// TwinCAT 3 PLC project PartDispencerPLC
// ProgramVersion: 3.1.4023.0
// libraries:
//   Tc2_MC2, * (Beckhoff Automation GmbH)
//   Tc2_NC, * (Beckhoff Automation GmbH)
//   Tc2_Standard, * (Beckhoff Automation GmbH)
//   Tc2_System, * (Beckhoff Automation GmbH)
//   Tc3_Module, * (Beckhoff Automation GmbH)
// project tree:
//   DUTs/ ST_StationControls.TcDUT
//   GVLs/ Globals.TcGVL, IO.TcGVL
//   / PlcTask.TcTTO
//   POUs/Conveyor/ FB_Conveyor.TcPOU
//   POUs/ MAIN.TcPOU
//   POUs/StationBin/ FB_StationBin.TcPOU
// real-time tasks:
//   TASK PlcTask: cycle T#10ms, priority 20, ADS port 350
// motion (NC):
//   TASK NC-Task 1 SAF: cycle T#2ms, priority 4, ADS port 501
//   TASK NC-Task 1 SVB: cycle T#10ms, priority 8, ADS port 511
//   AXIS Axis Ref (id 1)
//     OtherSettings: AllowMotionCmdToSlave=true
//     encoder EncType=4
//       EncPara: MaxCount=#x0000ffff
//         Inc: RefSoftSyncMask=#x0000ffff
//     drive DrvType=5
//       Analog: TorqueSetpointScale=10, ScaleFactorActTorque=0.1
//       TimeComp: TaskDelayCycles=1
//     controller CtrType=1
//       CtrPara: PriorControlFactor=1
//         Observer: BandWidth=20
// I/O:
//   DEVICE Device 1 (EtherCAT) (disabled), AmsNetId 192.168.0.103.2.1
//     Term 1 (EK1100) [EK1100 EtherCAT Coupler (2A E-Bus)]
//       Term 2 (EL1809) [EL1809 16Ch. Dig. Input 24V, 3ms]
//       Term 3 (EL1809) [EL1809 16Ch. Dig. Input 24V, 3ms]
//       Term 4 (EL2809) [EL2809 16Ch. Dig. Output 24V, 0.5A]
//       Term 5 (EL2809) [EL2809 16Ch. Dig. Output 24V, 0.5A]
//       Term 6 (EL2521) [EL2521 1Ch. Pulse Train Output]
// variable links:
//   NC-Task 1 SAF/Axes/Axis Ref <-> Device 1 (EtherCAT)/Term 1 (EK1100)/Term 6 (EL2521)
//     Drive/Inputs/In/nState1 @bit 6 <-> PTO Status/Status/Error
//     Drive/Inputs/In/nState1 @bit 1 <-> PTO Status/Status/Ramp active
//     Drive/Inputs/In/nState1 <-> PTO Status/Status/Sel. Ack/End counter
//     Drive/Inputs/In/nState1 @bit 4 <-> PTO Status/Status/Status of input target
//     Drive/Inputs/In/nState1 @bit 5 <-> PTO Status/Status/Status of input zero
//     Drive/Inputs/In/nState2 @bit 5 <-> PTO Status/Status/Sync error
//     Drive/Inputs/In/nState2 @bit 7 <-> PTO Status/Status/TxPDO Toggle
//     Drive/Inputs/In/nState4 @bit 1 <-> WcState/InputToggle
//     Drive/Inputs/In/nState4 <-> WcState/WcState
//     Drive/Outputs/Out/nCtrl1 @bit 1 <-> PTO Control/Control/Disable ramp
//     Drive/Outputs/Out/nCtrl1 <-> PTO Control/Control/Frequency select
//     Drive/Outputs/Out/nCtrl1 @bit 2 <-> PTO Control/Control/Go counter
//     Drive/Outputs/Out/nDataOut1[0] <-> PTO Control/Frequency value
//     Drive/Outputs/Out/nDataOut5 <-> PTO Target compact/Target counter value
//     Enc/Inputs/In/nDataIn1[0] <-> ENC Status compact/Counter value
//     Enc/Inputs/In/nState1 @bit 4 <-> ENC Status compact/Status/Counter overflow
//     Enc/Inputs/In/nState1 @bit 3 <-> ENC Status compact/Status/Counter underflow
//     Enc/Inputs/In/nState1 @bit 2 <-> ENC Status compact/Status/Set counter done
//     Enc/Inputs/In/nState2 @bit 5 <-> ENC Status compact/Status/Sync error
//     Enc/Inputs/In/nState2 @bit 7 <-> ENC Status compact/Status/TxPDO Toggle
//     Enc/Inputs/In/nState4 @bit 1 <-> WcState/InputToggle
//     Enc/Inputs/In/nState4 <-> WcState/WcState
//     Enc/Outputs/Out/nCtrl1 @bit 2 <-> ENC Control compact/Control/Set counter
//     Enc/Outputs/Out/nDataOut1[0] <-> ENC Control compact/Set counter value
//   PartDispencerPLC/PartDispencerPLC Instance <-> Device 1 (EtherCAT)/Term 1 (EK1100)/Term 2 (EL1809)
//     PlcTask Inputs/IO.iBowl_present_sensor_on_clamp <-> Channel 16/Input
//     PlcTask Inputs/IO.iStation_1_1_Dispense_Sensor <-> Channel 3/Input
//     PlcTask Inputs/IO.iStation_1_2_Dispense_Sensor <-> Channel 6/Input
//     PlcTask Inputs/IO.iStation_1_3_Dispense_Sensor <-> Channel 9/Input
//     PlcTask Inputs/IO.iStation_2_1_Dispense_Sensor <-> Channel 12/Input
//     PlcTask Inputs/IO.iStation_2_2_Dispense_Sensor <-> Channel 15/Input
//     PlcTask Inputs/IO.iStation_1_1_Home_Sensor <-> Channel 1/Input
//     PlcTask Inputs/IO.iStation_1_2_Home_Sensor <-> Channel 4/Input
//     PlcTask Inputs/IO.iStation_1_3_Home_Sensor <-> Channel 7/Input
//     PlcTask Inputs/IO.iStation_2_1_Home_Sensor <-> Channel 10/Input
//     PlcTask Inputs/IO.iStation_2_2_Home_Sensor <-> Channel 13/Input
//     PlcTask Inputs/IO.iStation_1_1_Safe_Sensor <-> Channel 2/Input
//     PlcTask Inputs/IO.iStation_1_2_Safe_Sensor <-> Channel 5/Input
//     PlcTask Inputs/IO.iStation_1_3_Safe_Sensor <-> Channel 8/Input
//     PlcTask Inputs/IO.iStation_2_1_Safe_Sensor <-> Channel 11/Input
//     PlcTask Inputs/IO.iStation_2_2_Safe_Sensor <-> Channel 14/Input
//   PartDispencerPLC/PartDispencerPLC Instance <-> Device 1 (EtherCAT)/Term 1 (EK1100)/Term 3 (EL1809)
//     PlcTask Inputs/IO.iBowl_10_percent_full <-> Channel 10/Input
//     PlcTask Inputs/IO.iBowl_25_percent_full <-> Channel 9/Input
//     PlcTask Inputs/IO.iBowl_50_percent_full <-> Channel 8/Input
//     PlcTask Inputs/IO.iConveyor_Home_Sensor <-> Channel 4/Input
//     PlcTask Inputs/IO.iConveyor_Position_1_Sensor <-> Channel 5/Input
//     PlcTask Inputs/IO.iConveyor_Position_2_Sensor <-> Channel 6/Input
//     PlcTask Inputs/IO.iConveyor_Position_3_Sensor <-> Channel 7/Input
//     PlcTask Inputs/IO.iStation_1_1_Part_Present_Sensor <-> Channel 11/Input
//     PlcTask Inputs/IO.iStation_1_2_Part_Present_Sensor <-> Channel 12/Input
//     PlcTask Inputs/IO.iStation_1_3_Part_Present_Sensor <-> Channel 13/Input
//     PlcTask Inputs/IO.iStation_2_1_Part_Present_Sensor <-> Channel 14/Input
//     PlcTask Inputs/IO.iStation_2_2_Part_Present_Sensor <-> Channel 15/Input
//     PlcTask Inputs/IO.iStation_2_3_Part_Present_Sensor <-> Channel 16/Input
//     PlcTask Inputs/IO.iStation_2_3_Dispense_Sensor <-> Channel 3/Input
//     PlcTask Inputs/IO.iStation_2_3_Home_Sensor <-> Channel 1/Input
//     PlcTask Inputs/IO.iStation_2_3_Safe_Sensor <-> Channel 2/Input
//   PartDispencerPLC/PartDispencerPLC Instance <-> Device 1 (EtherCAT)/Term 1 (EK1100)/Term 4 (EL2809)
//     PlcTask Outputs/IO.oDirection_OF_Driver_1 <-> Channel 2/Output
//     PlcTask Outputs/IO.oDirection_of_Driver_{2..5} <-> Channel {5..14 step 3}/Output  (4 links)
//     PlcTask Outputs/IO.oEnable_of_Driver_{1..5} <-> Channel {3..15 step 3}/Output  (5 links)
//     PlcTask Outputs/IO.oR{1..5}_NO_Contact <-> Channel {1..13 step 3}/Output  (5 links)
//     PlcTask Outputs/IO.oSPARE_1 <-> Channel 16/Output
//   PartDispencerPLC/PartDispencerPLC Instance <-> Device 1 (EtherCAT)/Term 1 (EK1100)/Term 5 (EL2809)
//     PlcTask Outputs/IO.oDirection_OF_Driver_6 <-> Channel 2/Output
//     PlcTask Outputs/IO.oDirection_of_Driver_7 <-> Channel 5/Output
//     PlcTask Outputs/IO.oDirection_of_Driver_8 <-> Channel 8/Output
//     PlcTask Outputs/IO.oEnable_of_Driver_6 <-> Channel 3/Output
//     PlcTask Outputs/IO.oEnable_of_Driver_7 <-> Channel 6/Output
//     PlcTask Outputs/IO.oEnable_of_Driver_8 <-> Channel 9/Output
//     PlcTask Outputs/IO.oR6_NO_Contact <-> Channel 1/Output
//     PlcTask Outputs/IO.oR7_NO_Contact <-> Channel 4/Output
//     PlcTask Outputs/IO.oR8_NO_Contact <-> Channel 7/Output
//     PlcTask Outputs/IO.oSPARE_{5..11} <-> Channel {10..16}/Output  (7 links)

CONFIGURATION PartDispencerPLC
    RESOURCE PLC ON TwinCAT3
        TASK PlcTask(INTERVAL := T#10ms, PRIORITY := 20);
        PROGRAM MAIN WITH PlcTask : MAIN;
    END_RESOURCE
END_CONFIGURATION

// ---- DUTs/ST_StationControls.TcDUT
TYPE ST_StationControls :
STRUCT
	bEnable			: BOOL;
	bReset			: BOOL;
	bError			: BOOL;
	sStatus			: STRING(255);
END_STRUCT
END_TYPE

// ---- GVLs/Globals.TcGVL
{attribute 'qualified_only'}
VAR_GLOBAL
	ConveyorControl			:ST_StationControls;
	
	Bin1Control				:ST_StationControls;
	Bin2Control				:ST_StationControls;
	Bin3Control				:ST_StationControls;
	Bin4Control				:ST_StationControls;
	Bin5Control				:ST_StationControls;
	Bin6Control				:ST_StationControls;
	
	bResetPartCount_Station1	: BOOL := FALSE;
	bResetPartCount_Station2	: BOOL := FALSE;
	
	axisRef						: AXIS_REF;
END_VAR

// ---- GVLs/IO.TcGVL
{attribute 'qualified_only'}
VAR_GLOBAL
// ======================== Inputs ==================================
	// SLOT 1 - EL1809
	iStation_1_1_Home_Sensor				AT %I* :BOOL;
	iStation_1_1_Safe_Sensor             	AT %I* :BOOL;
	iStation_1_1_Dispense_Sensor         	AT %I* :BOOL;
	iStation_1_2_Home_Sensor             	AT %I* :BOOL;
	iStation_1_2_Safe_Sensor             	AT %I* :BOOL;
	iStation_1_2_Dispense_Sensor         	AT %I* :BOOL;
	iStation_1_3_Home_Sensor             	AT %I* :BOOL;
	iStation_1_3_Safe_Sensor             	AT %I* :BOOL;
	iStation_1_3_Dispense_Sensor         	AT %I* :BOOL;
	iStation_2_1_Home_Sensor             	AT %I* :BOOL;
	iStation_2_1_Safe_Sensor             	AT %I* :BOOL;
	iStation_2_1_Dispense_Sensor         	AT %I* :BOOL;
	iStation_2_2_Home_Sensor             	AT %I* :BOOL;
	iStation_2_2_Safe_Sensor             	AT %I* :BOOL;
	iStation_2_2_Dispense_Sensor         	AT %I* :BOOL;
	iBowl_present_sensor_on_clamp			AT %I* :BOOL;

	// SLOT 2 - EL1809
	iStation_2_3_Home_Sensor				AT %I* :BOOL;
	iStation_2_3_Safe_Sensor             	AT %I* :BOOL;
	iStation_2_3_Dispense_Sensor         	AT %I* :BOOL;
	iConveyor_Home_Sensor                	AT %I* :BOOL; 
	iConveyor_Position_1_Sensor				AT %I* :BOOL; 	// Staion 1
	iConveyor_Position_2_Sensor				AT %I* :BOOL;	// Station 2
	iConveyor_Position_3_Sensor				AT %I* :BOOL;	// Collection point
	iBowl_50_percent_full					AT %I* :BOOL;
	iBowl_25_percent_full					AT %I* :BOOL;
	iBowl_10_percent_full					AT %I* :BOOL;
	iStation_1_1_Part_Present_Sensor		AT %I* :BOOL;
	iStation_1_2_Part_Present_Sensor		AT %I* :BOOL;
	iStation_1_3_Part_Present_Sensor        AT %I* :BOOL;
	iStation_2_1_Part_Present_Sensor        AT %I* :BOOL;
	iStation_2_2_Part_Present_Sensor        AT %I* :BOOL;
	iStation_2_3_Part_Present_Sensor        AT %I* :BOOL;

// ======================== Outputs ==================================
	// Slot 3 - EL2809
	oR1_NO_Contact							AT %Q* :BOOL;
	oDirection_OF_Driver_1                  AT %Q* :BOOL;
	oEnable_of_Driver_1                     AT %Q* :BOOL;
	oR2_NO_Contact                          AT %Q* :BOOL;
	oDirection_of_Driver_2                  AT %Q* :BOOL;
	oEnable_of_Driver_2                     AT %Q* :BOOL;
	oR3_NO_Contact                          AT %Q* :BOOL;
	oDirection_of_Driver_3                  AT %Q* :BOOL;
	oEnable_of_Driver_3                     AT %Q* :BOOL;
	oR4_NO_Contact                          AT %Q* :BOOL;
	oDirection_of_Driver_4                  AT %Q* :BOOL;
	oEnable_of_Driver_4                     AT %Q* :BOOL;
	oR5_NO_Contact                          AT %Q* :BOOL;
	oDirection_of_Driver_5                  AT %Q* :BOOL;
	oEnable_of_Driver_5                     AT %Q* :BOOL;
	oSPARE_1                                AT %Q* :BOOL;
	
	// SLot 4 - EL2809
	oR6_NO_Contact							AT %Q* :BOOL;
	oDirection_OF_Driver_6                  AT %Q* :BOOL;
	oEnable_of_Driver_6                     AT %Q* :BOOL;
	oR7_NO_Contact 							AT %Q* :BOOL;				//(Conveyor)
	oDirection_of_Driver_7  				AT %Q* :BOOL;				//(Conveyor)
	oEnable_of_Driver_7  					AT %Q* :BOOL;				//(Conveyor)
	oR8_NO_Contact 			                AT %Q* :BOOL;
	oDirection_of_Driver_8                  AT %Q* :BOOL;
	oEnable_of_Driver_8  	                AT %Q* :BOOL;
	oSPARE_5                                AT %Q* :BOOL;
	oSPARE_6                                AT %Q* :BOOL;
	oSPARE_7                                AT %Q* :BOOL;
	oSPARE_8                                AT %Q* :BOOL;
	oSPARE_9                                AT %Q* :BOOL;
	oSPARE_10                               AT %Q* :BOOL;
	oSPARE_11                               AT %Q* :BOOL;


END_VAR

// ---- POUs/MAIN.TcPOU
PROGRAM MAIN
VAR
	//Conveyor
	Conveyor		: FB_Conveyor;
	
	// Station 1
	Station1_Bin1	: FB_StationBin;
	Station1_Bin2	: FB_StationBin;
	Station1_Bin3	: FB_StationBin;
	
	//Station 2
	Station2_Bin1	: FB_StationBin;
	Station2_Bin2	: FB_StationBin;
	Station2_Bin3	: FB_StationBin;
	
	// Stations Ready
	bStation1_Ready : BOOL;
	bStation2_Ready : BOOL;
	
	// Reset Bins
	bResetCount_Bin1: BOOL;
	bResetCount_Bin2: BOOL;
	bResetCount_Bin3: BOOL;
	bResetCount_Bin4: BOOL;
	bResetCount_Bin5: BOOL;
	bResetCount_Bin6: BOOL;
END_VAR

a_EnableDrives();

Conveyor(
	Station_1_Ready:= bStation1_Ready, 
	Station_2_Ready:= bStation2_Ready, 
	At_Station_1=> , 
	At_Station_2=> , 
	At_Station_3=> , 
	ResetConvoyor := Globals.ConveyorControl.bReset,
	sStatus=> Globals.ConveyorControl.sStatus, 
	bError=> Globals.ConveyorControl.bError);
	
Station1_Bin1(
	bEnableBin := Globals.Bin1Control.bEnable,
	Home_Sensor:= IO.iStation_1_1_Home_Sensor, 
	Safe_Sensor:= IO.iStation_1_1_Safe_Sensor, 
	Dispense_Sensor:= IO.iStation_1_1_Dispense_Sensor, 
	Part_Present := IO.iStation_1_1_Part_Present_Sensor,
	Dependency_OK:= NOT Station1_Bin2.Lock_Dependency AND NOT Station1_Bin3.Lock_Dependency, 
	At_Station:= Conveyor.At_Station_1, 
	Trigger_OF_Drive=> IO.oR1_NO_Contact, 
	Direction_OF_Drive=> IO.oDirection_OF_Driver_1, 
	Lock_Dependency=> , 
	ResetPartCount := bResetCount_Bin1,
	ResetBin := Globals.Bin1Control.bReset,
	bError=> Globals.Bin1Control.bError, 
	sStatus=> Globals.Bin1Control.sStatus);
	
Station1_Bin2(
	bEnableBin := Globals.Bin2Control.bEnable,
	Home_Sensor:= IO.iStation_1_2_Home_Sensor, 
	Safe_Sensor:= IO.iStation_1_2_Safe_Sensor, 
	Dispense_Sensor:= IO.iStation_1_2_Dispense_Sensor,
	Part_Present := IO.iStation_1_2_Part_Present_Sensor, 
	Dependency_OK:= NOT Station1_Bin1.Lock_Dependency AND NOT Station1_Bin3.Lock_Dependency, 
	At_Station:= Conveyor.At_Station_1, 
	Trigger_OF_Drive=> IO.oR2_NO_Contact, 
	Direction_OF_Drive=> IO.oDirection_OF_Driver_2, 
	Lock_Dependency=> , 
	ResetPartCount := bResetCount_Bin2,
	ResetBin := Globals.Bin2Control.bReset,
	bError=> Globals.Bin2Control.bError , 
	sStatus=> Globals.Bin2Control.sStatus);
	
Station1_Bin3(
	bEnableBin := Globals.Bin3Control.bEnable,
	Home_Sensor:= IO.iStation_1_3_Home_Sensor, 
	Safe_Sensor:= IO.iStation_1_3_Safe_Sensor, 
	Dispense_Sensor:= IO.iStation_1_3_Dispense_Sensor,
	Part_Present := IO.iStation_1_3_Part_Present_Sensor, 
	Dependency_OK:= NOT Station1_Bin1.Lock_Dependency AND NOT Station1_Bin2.Lock_Dependency, 
	At_Station:= Conveyor.At_Station_1, 
	Trigger_OF_Drive=> IO.oR3_NO_Contact, 
	Direction_OF_Drive=> IO.oDirection_OF_Driver_3, 
	Lock_Dependency=> , 
	ResetPartCount := bResetCount_Bin3,
	ResetBin := Globals.Bin3Control.bReset,
	bError=> Globals.Bin3Control.bError, 
	sStatus=> Globals.Bin3Control.sStatus);
	
Station2_Bin1(
	bEnableBin := Globals.Bin4Control.bEnable,
	Home_Sensor:= IO.iStation_2_1_Home_Sensor, 
	Safe_Sensor:= IO.iStation_2_1_Safe_Sensor, 
	Dispense_Sensor:= IO.iStation_2_1_Dispense_Sensor,
	Part_Present := IO.iStation_2_1_Part_Present_Sensor, 
	Dependency_OK:= NOT Station2_Bin2.Lock_Dependency AND NOT Station2_Bin3.Lock_Dependency, 
	At_Station:= Conveyor.At_Station_2, 
	Trigger_OF_Drive=> IO.oR4_NO_Contact, 
	Direction_OF_Drive=> IO.oDirection_OF_Driver_4, 
	Lock_Dependency=> , 
	ResetPartCount := bResetCount_Bin4,
	ResetBin := Globals.Bin4Control.bReset,
	bError=>Globals.Bin4Control.bError , 
	sStatus=> Globals.Bin4Control.sStatus);
	
Station2_Bin2(
	bEnableBin := Globals.Bin5Control.bEnable,
	Home_Sensor:= IO.iStation_2_2_Home_Sensor, 
	Safe_Sensor:= IO.iStation_2_2_Safe_Sensor, 
	Dispense_Sensor:= IO.iStation_2_2_Dispense_Sensor, 
	Part_Present := IO.iStation_2_2_Part_Present_Sensor,
	Dependency_OK:= NOT Station2_Bin1.Lock_Dependency AND NOT Station2_Bin3.Lock_Dependency, 
	At_Station:= Conveyor.At_Station_2, 
	Trigger_OF_Drive=> IO.oR5_NO_Contact, 
	Direction_OF_Drive=> IO.oDirection_OF_Driver_5, 
	Lock_Dependency=> , 
	ResetPartCount := bResetCount_Bin5,
	ResetBin := Globals.Bin5Control.bReset,
	bError=> Globals.Bin5Control.bError, 
	sStatus=> Globals.Bin5Control.sStatus);
	
Station2_Bin3(
	bEnableBin := Globals.Bin6Control.bEnable,
	Home_Sensor:= IO.iStation_2_3_Home_Sensor, 
	Safe_Sensor:= IO.iStation_2_3_Safe_Sensor, 
	Dispense_Sensor:= IO.iStation_2_3_Dispense_Sensor,
	Part_Present := IO.iStation_2_3_Part_Present_Sensor, 
	Dependency_OK:= NOT Station2_Bin1.Lock_Dependency AND NOT Station2_Bin2.Lock_Dependency, 
	At_Station:= Conveyor.At_Station_2, 
	Trigger_OF_Drive=> IO.oR6_NO_Contact, 
	Direction_OF_Drive=> IO.oDirection_OF_Driver_6, 
	Lock_Dependency=> , 
	ResetPartCount := bResetCount_Bin6,
	ResetBin := Globals.Bin6Control.bReset,
	bError=> Globals.Bin6Control.bError, 
	sStatus=> Globals.Bin6Control.sStatus);
	
// Ready Conditions
bStation1_Ready := Station1_Bin1.Count_OF_Parts + Station1_Bin2.Count_OF_Parts + Station1_Bin3.Count_OF_Parts >= 15;
bStation2_Ready := Station2_Bin1.Count_OF_Parts + Station2_Bin2.Count_OF_Parts + Station2_Bin3.Count_OF_Parts >= 15;
IF Globals.bResetPartCount_Station1 
AND (Station1_Bin1.Count_OF_Parts + Station1_Bin2.Count_OF_Parts + Station1_Bin3.Count_OF_Parts > 0) THEN
	bResetCount_Bin1:= TRUE;
	bResetCount_Bin2:= TRUE;
	bResetCount_Bin3:= TRUE;
ELSE
	Globals.bResetPartCount_Station1 := FALSE;
END_IF

IF Globals.bResetPartCount_Station2 
AND (Station2_Bin1.Count_OF_Parts + Station2_Bin2.Count_OF_Parts + Station2_Bin3.Count_OF_Parts > 0) THEN
	bResetCount_Bin4 := TRUE;
	bResetCount_Bin5 := TRUE;
	bResetCount_Bin6 := TRUE;
ELSE
	Globals.bResetPartCount_Station2 := FALSE;
END_IF

ACTION a_EnableDrives:
IO.oEnable_of_Driver_1 := TRUE;
IO.oEnable_of_Driver_2 := TRUE;
IO.oEnable_of_Driver_3 := TRUE;
IO.oEnable_of_Driver_4 := TRUE;
IO.oEnable_of_Driver_5 := TRUE;
IO.oEnable_of_Driver_6 := TRUE;
IO.oEnable_of_Driver_7 := TRUE;
IO.oEnable_of_Driver_8 := TRUE;
END_ACTION

END_PROGRAM

// ---- POUs/Conveyor/FB_Conveyor.TcPOU
FUNCTION_BLOCK FB_Conveyor
VAR_INPUT
	Station_1_Ready : BOOL;
	Station_2_Ready : BOOL;
END_VAR

VAR_OUTPUT
	At_Station_1	: BOOL;
	At_Station_2	: BOOL;
	At_Station_3	: BOOL;
	sStatus			: STRING(255);
	bError			: BOOL;
END_VAR
VAR_IN_OUT
	ResetConvoyor		: BOOL;						// Reset Conveyor Logic
END_VAR
VAR
	TimerTimeout		: TON;						// Used for Timeouts
	
	// Times
	tTimeoutMoving		: TIME := T#5000MS; 		// Timeout When Stepper motor moving between positions
	tTimeoutBowlLoading	: TIME := T#5000MS;			//
	
	iStep				: INT; 						// Step of machine logic
	iStepClamp			: INT;
	bLoadBowl			: BOOL;
	bBowlLoaded			: BOOL;
END_VAR

a_LoadBowl();
IF ResetConvoyor THEN
	iStep := 0;
	IO.oR7_NO_Contact := FALSE;
END_IF
CASE iStep OF 
	0: // Start Bowl Loading
		IF bError THEN
			bError := FALSE;
		END_IF
		IF NOT Station_1_Ready
		AND NOT Station_2_Ready
		THEN
			IF NOT IO.iConveyor_Home_Sensor
			AND NOT IO.iConveyor_Position_1_Sensor
			AND NOT IO.iConveyor_Position_2_Sensor 
			AND NOT IO.iConveyor_Position_3_Sensor
			THEN
				iStep := 10;
			ELSIF IO.iConveyor_Home_Sensor
			AND NOT IO.iConveyor_Position_1_Sensor 
			AND NOT IO.iConveyor_Position_2_Sensor
			AND NOT IO.iConveyor_Position_3_Sensor
			THEN
				iStep := 20;	
			ELSIF NOT IO.iConveyor_Home_Sensor
			AND IO.iConveyor_Position_1_Sensor 
			AND NOT IO.iConveyor_Position_2_Sensor
			AND NOT IO.iConveyor_Position_3_Sensor
			THEN
				iStep := 10;
			ELSIF IO.iConveyor_Home_Sensor
			AND IO.iConveyor_Position_1_Sensor 
			AND NOT IO.iConveyor_Position_2_Sensor
			AND NOT IO.iConveyor_Position_3_Sensor
			THEN
				iStep := 20;
			ELSIF NOT IO.iConveyor_Home_Sensor
			AND IO.iConveyor_Position_1_Sensor 
			AND IO.iConveyor_Position_2_Sensor
			AND NOT IO.iConveyor_Position_3_Sensor
			THEN
				iStep := 30;
			ELSIF IO.iConveyor_Position_3_Sensor THEN
				sStatus := 'Waiting Remove the Bowl on station 3';
			END_IF	
		ELSE
			iStep := 40;
		END_IF
// ======================= Start Cycle =====================================		
	10: //Wait Bowl Loadin Start
		bLoadBowl := TRUE;
		sStatus := 'Loading Bowl on Conveyor Home';
		IF NOT bBowlLoaded
		AND iStepClamp > 0 THEN
			iStep := 2;
		END_IF
	
	11: // Wait Bowl on Conveyor
		IF NOT bLoadBowl
		AND bBowlLoaded THEN
			iStep := 0;
		END_IF
		
	20: // Start Send Bowl to Station 1 
		sStatus := 'Moving Bowls';
		IO.oR7_NO_Contact := TRUE;
		IO.oDirection_of_Driver_7 := TRUE;
		iStep := 11;
		
	21: // Wait Send Bowl to Station 1
		TimerTimeout(IN := TRUE, PT:= tTimeoutMoving);
		IF IO.iConveyor_Position_1_Sensor
		AND NOT IO.iConveyor_Position_2_Sensor THEN
			IO.oR7_NO_Contact := FALSE;
			TimerTimeout(IN := FALSE);
			iStep := 0;
		ELSIF IO.iConveyor_Position_1_Sensor
		AND IO.iConveyor_Position_2_Sensor THEN
			IO.oR7_NO_Contact := FALSE;
			TimerTimeout(IN := FALSE);
			iStep := 0;
		ELSIF TimerTimeout.Q THEN
			sStatus := 'Timeout When Going to Position 1';
			iStep := 1000; // Error
		END_IF
// ======================= Wait Stations Ready =============================				
	30: // Wait Stations Ready
		At_Station_1 := NOT Station_1_Ready;
		At_Station_2 := NOT Station_2_Ready;
		sStatus := 'Waiting for Stations Ready';
		IF Station_1_Ready 
		AND Station_2_Ready THEN
			iStep := 40;
		END_IF
// ======================= End Cycle =====================================		
	40: // Check End Cylce Conditions
		sStatus := 'Checking End Cycle Conditions';
		IF NOT IO.iConveyor_Home_Sensor
		AND IO.iConveyor_Position_1_Sensor 
		AND IO.iConveyor_Position_2_Sensor
		AND NOT IO.iConveyor_Position_3_Sensor
		THEN			
			iStep := 50;
		ELSIF NOT IO.iConveyor_Home_Sensor
		AND NOT IO.iConveyor_Position_1_Sensor 
		AND IO.iConveyor_Position_2_Sensor
		AND NOT IO.iConveyor_Position_3_Sensor
		THEN	
			iStep := 50;
		ELSIF NOT IO.iConveyor_Home_Sensor
		AND NOT IO.iConveyor_Position_1_Sensor 
		AND NOT IO.iConveyor_Position_2_Sensor
		AND NOT IO.iConveyor_Position_3_Sensor
		THEN	
			iStep := 70;
		ELSIF IO.iConveyor_Position_3_Sensor THEN
			sStatus := 'Waiting Remove the Bowl on station 3';
		END_IF
		
	50: // Start Moving Full Bowl to Station 3
		sStatus := 'Moving Bowl 1 End Cycle';
		IO.oR7_NO_Contact := TRUE;
		IO.oDirection_of_Driver_7 := TRUE;
		iStep := 51;
	
	51: // Wait on Station 3
		TimerTimeout(IN := TRUE, PT:= tTimeoutMoving);
		IF IO.iConveyor_Position_3_Sensor THEN
			IO.oR7_NO_Contact := FALSE;
			TimerTimeout(IN := FALSE);
			iStep := 60;
		ELSIF TimerTimeout.Q THEN
			sStatus := 'Timeout When Going to Position 3';
			iStep := 1000; // Error
		END_IF
		
	60:// Wait remove Bowl Station 3
		sStatus := 'Waiting Remove the Bowl on station 3';
		IF NOT IO.iConveyor_Position_3_Sensor THEN
			iStep := 40;
		END_IF		
		
	70: //Start Reset Counters
		Globals.bResetPartCount_Station1 := TRUE;
		Globals.bResetPartCount_Station2 := TRUE;
		iStep := 71;
		
	71: // Wait Reset Counters
		sStatus := 'Waiting Part Counter Reset';
		IF NOT Station_1_Ready
		AND NOT Station_2_Ready
		AND NOT Globals.bResetPartCount_Station1
		AND NOT Globals.bResetPartCount_Station2
		THEN
			iStep := 0;
		END_IF
	
	1000: // ERROR
		TimerTimeout(IN := FALSE);
		bError := TRUE;
		IO.oR7_NO_Contact := FALSE;
END_CASE

ACTION a_LoadBowl:
IF NOT bLoadBowl THEN
	iStepClamp := 0;
	IO.oR8_NO_Contact := FALSE;
ELSE
	CASE iStepClamp OF
		0: // Wait Bowls in clamp
			IF NOT IO.iBowl_10_percent_full THEN
				sStatus := 'Bowls in clamp under 10 percent!';
			ELSE
				bBowlLoaded := FALSE;
				iStepClamp := 1;
			END_IF
			
		1: // Check Bowl on Home
			IF NOT IO.iConveyor_Home_Sensor THEN
				iStepClamp := 10;
			ELSE
				iStepClamp := 30;
			END_IF
			
		10: //Start Open Clamp
			IO.oR8_NO_Contact := TRUE;
			IO.oDirection_of_Driver_8 := TRUE;
			iStepClamp := 20;
			
		20:
			// Wait Bowl on Conveyor
			TimerTimeout(IN:= TRUE, PT := tTimeoutBowlLoading);
			IF IO.iConveyor_Home_Sensor THEN
				TimerTimeout(IN:= FALSE);
				IO.oR8_NO_Contact := FALSE;
				iStepClamp := 30;
			ELSIF TimerTimeout.Q THEN
				sStatus := 'Timeout: Bowl not in Conveyor Home!';
				iStep := 1000;
			END_IF
		
		30: // End
			bLoadBowl := FALSE;
			bBowlLoaded := TRUE;
	END_CASE
END_IF
END_ACTION

END_FUNCTION_BLOCK

// ---- POUs/StationBin/FB_StationBin.TcPOU
FUNCTION_BLOCK FB_StationBin
VAR_INPUT
	bEnableBin			: BOOL; // input for Enable Bin 
	Home_Sensor 		: BOOL; // input for home
	Safe_Sensor 		: BOOL;	// input for safe
	Dispense_Sensor 	: BOOL; // input for dispense
	Part_Present		: BOOL; // input for part present
	Dependency_OK		: BOOL; // input to check for dependency
	At_Station			: BOOL; // Input for bowl at station, used for reset condition too
END_VAR
VAR_OUTPUT
	Trigger_Of_Drive	: BOOL;	// Output for Enable of drive movement
	Direction_OF_Drive	: BOOL; // Output for Direction of drive - TRUE- Direction Positive, False - Direction Negative
	Lock_Dependency		: BOOL; // Output for Lock Dependency
	Count_OF_Parts		: INT;	// Counting of loaded parts
	bError				: BOOL; // Station is in Error
	sStatus				: STRING(255); // Message
END_VAR
VAR_IN_OUT
	ResetPartCount		: BOOL;		// Reset Counter of parts
	ResetBin			: BOOL;		// Reset Bin Logic
END_VAR
VAR
	TimerTimeout		: TON; // Use for timeout
	
	// Times
	tTimeoutMoving		: TIME := T#5000MS;
	tTimeoutDispence	: TIME := T#2000MS;
	
	iStep				: INT; // Step of the machine logic
END_VAR

IF NOT bEnableBin THEN
	iStep := 0;
	bError := FALSE;
	sStatus := 'Waiting for bin Enable';
	Count_OF_Parts := 0;
	Lock_Dependency := FALSE;
	Trigger_Of_Drive := FALSE;
ELSE
	IF ResetPartCount THEN
		ResetPartCount := FALSE;
		Count_OF_Parts := 0;
	END_IF
	IF ResetBin THEN
		ResetBin := FALSE;
		iStep := 0;
		Count_OF_Parts := 0;
		Lock_Dependency := FALSE;
		Trigger_Of_Drive := FALSE;
	END_IF
	CASE iStep OF
		0:  // Waiting part on Home
			IF bError THEN
				bError := FALSE;
			END_IF
			sStatus := 'Waiting for Part on Home';
			IF Home_Sensor 
			AND Part_Present 
			THEN
				iStep := 10;
			END_IF
			
		10: // Move to Safe
			Trigger_Of_Drive := TRUE;
			Direction_OF_Drive := TRUE;
			iStep := 11;
			
		11: // Wait Safe Done
			TimerTimeout(IN := TRUE, PT:= tTimeoutMoving);
			IF Safe_Sensor THEN
				Trigger_Of_Drive := FALSE;
				TimerTimeout(IN := FALSE);
				iStep := 20;
			ELSIF TimerTimeout.Q THEN
				sStatus := 'Timeout When Going to Safe';
				iStep := 1000; // Error
			END_IF
		
		20: // Check Dependency OK
			sStatus := 'Waiting Dependency OK';
			IF Dependency_OK 
			AND AT_Station 
			THEN
				sStatus := 'Going to Dispense';
				Lock_Dependency := TRUE;
				iStep := 30;
			END_IF
		
		30: // Move to Dispense
			Trigger_Of_Drive := TRUE;
			Direction_OF_Drive := TRUE;
			iStep := 31;
			
		31: // Wait Dispense
			TimerTimeout(IN := TRUE, PT:= tTimeoutMoving);
			IF Dispense_Sensor THEN
				Trigger_Of_Drive := FALSE;
				TimerTimeout(IN := FALSE);
				iStep := 40;
			ELSIF TimerTimeout.Q THEN
				sStatus := 'Timeout When Going to Dispense';
				iStep := 1000; // Error
			END_IF
		
		40: // Check Dispense Done
			TimerTimeout(IN := TRUE, PT:= tTimeoutDispence);
			IF NOT Part_Present THEN
				Count_OF_Parts := Count_OF_Parts + 1;
				TimerTimeout(IN := FALSE);
				iStep := 50;
			ELSIF TimerTimeout.Q THEN
				sStatus := 'Timeout When Not Part Present - Dispense Done';
				iStep := 1000; // Error
			END_IF
			
		50: // Start Move back to Safety
			Trigger_Of_Drive := TRUE;
			Direction_OF_Drive := FALSE;
			iStep := 51;
			
		51: // Wait Move back to Safety
			TimerTimeout(IN := TRUE, PT:= tTimeoutMoving);
			IF Safe_Sensor THEN
				Trigger_Of_Drive := FALSE;
				Lock_Dependency := FALSE;
				TimerTimeout(IN := FALSE);
				iStep := 60;
			ELSIF TimerTimeout.Q THEN
				sStatus := 'Timeout When Going back to Safe';
				iStep := 1000; // Error
			END_IF
		
		60: // Start Move Back To Home
			Trigger_Of_Drive := TRUE;
			Direction_OF_Drive := FALSE;
			iStep := 61;
		
		61: // Wait Move Back to Home
			TimerTimeout(IN := TRUE, PT:= tTimeoutMoving);
			IF Home_Sensor THEN
				Trigger_Of_Drive := FALSE;
				TimerTimeout(IN := FALSE);
				iStep := 0;
			ELSIF TimerTimeout.Q THEN
				sStatus := 'Timeout When Going back to Safe';
				iStep := 1000; // Error
			END_IF	
			
		1000:
			bError := TRUE;
			Trigger_Of_Drive := FALSE;
			TimerTimeout(IN := FALSE);
	END_CASE
END_IF

END_FUNCTION_BLOCK
